// TIA Portal V21 export
FUNCTION_BLOCK "DoFb"   // FB109, LAD
{ S7_Optimized_Access := 'FALSE' }
// stored: AutoNumber false, SetENOAutomatically false
   VAR_INPUT
      sec : Bool;
      AlarmAck : Bool;
      AlwaysTrue : Bool;
      AlwaysFalse : Bool;
      Interlock : Bool;
   END_VAR
   VAR
      Do01 { S7_SetPoint := 'True'} : "DigitalOutput";   // Mm01Cmd
      Do02 { S7_SetPoint := 'True'} : "DigitalOutput";   // Cp01Cmd
      Do03 { S7_SetPoint := 'True'} : "DigitalOutput";   // Htr
      Do04 { S7_SetPoint := 'True'} : "DigitalOutput";   // Lf01
      Do05 { S7_SetPoint := 'True'} : "DigitalOutput";   // DoSpare1
      Do06 { S7_SetPoint := 'True'} : "DigitalOutput";   // DoSpare2
      Do07 { S7_SetPoint := 'True'} : "DigitalOutput";   // DoSpare3
      Do08 { S7_SetPoint := 'True'} : "DigitalOutput";   // DoSpare4
      Do09 { S7_SetPoint := 'True'} : "DigitalOutput";   // DoSpare5
      Do10 { S7_SetPoint := 'True'} : "DigitalOutput";   // DoSpare6
   END_VAR
BEGIN

REGION Network 1: Mm01Cmd
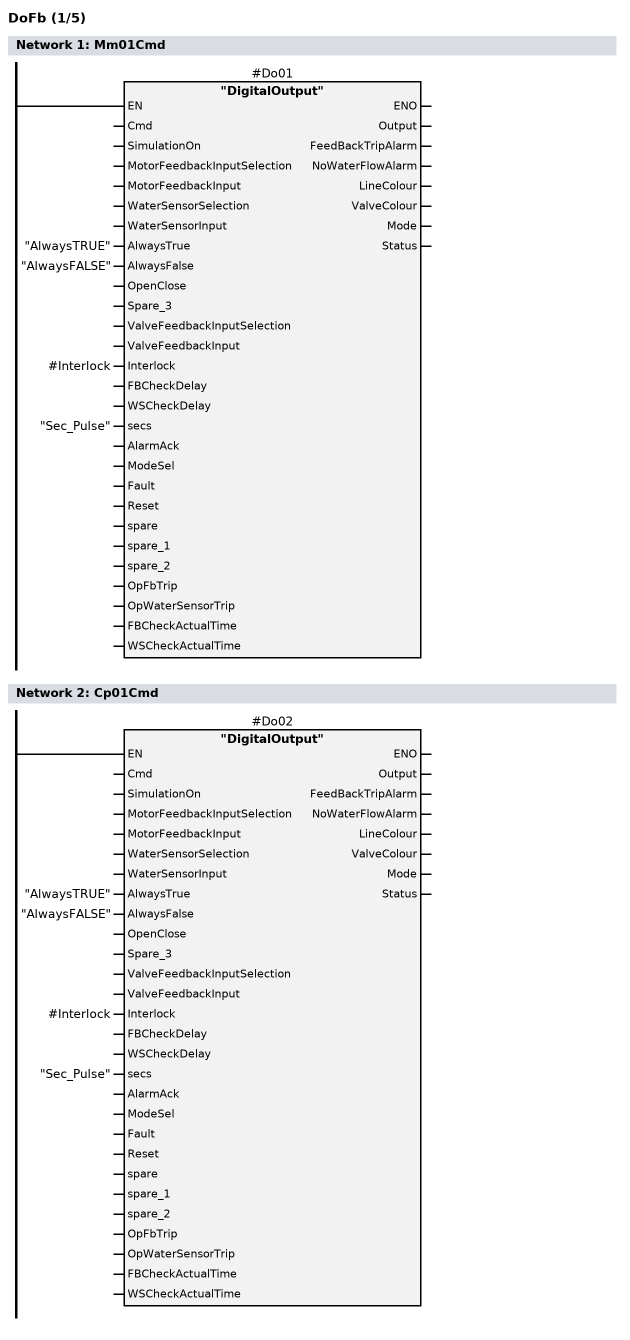
   RUNG wire#powerrail
      #Do01(Cmd :=, SimulationOn :=, MotorFeedbackInputSelection :=, MotorFeedbackInput :=, WaterSensorSelection :=, WaterSensorInput :=, AlwaysTrue := "AlwaysTRUE", AlwaysFalse := "AlwaysFALSE", OpenClose :=, Spare_3 :=, ValveFeedbackInputSelection :=, ValveFeedbackInput :=, Interlock := #Interlock, FBCheckDelay :=, WSCheckDelay :=, secs := "Sec_Pulse", AlarmAck :=, ModeSel :=, Fault :=, Reset :=, spare :=, spare_1 :=, spare_2 :=, OpFbTrip :=, OpWaterSensorTrip :=, FBCheckActualTime :=, WSCheckActualTime :=, Output =>, FeedBackTripAlarm =>, NoWaterFlowAlarm =>, LineColour =>, ValveColour =>, Mode =>, Status =>)
   END_RUNG
   // the same network as SCL:
   #Do01(AlwaysTrue := "AlwaysTRUE", AlwaysFalse := "AlwaysFALSE", Interlock := #Interlock, secs := "Sec_Pulse");   // "DigitalOutput"
END_REGION

REGION Network 2: Cp01Cmd
   RUNG wire#powerrail
      #Do02(Cmd :=, SimulationOn :=, MotorFeedbackInputSelection :=, MotorFeedbackInput :=, WaterSensorSelection :=, WaterSensorInput :=, AlwaysTrue := "AlwaysTRUE", AlwaysFalse := "AlwaysFALSE", OpenClose :=, Spare_3 :=, ValveFeedbackInputSelection :=, ValveFeedbackInput :=, Interlock := #Interlock, FBCheckDelay :=, WSCheckDelay :=, secs := "Sec_Pulse", AlarmAck :=, ModeSel :=, Fault :=, Reset :=, spare :=, spare_1 :=, spare_2 :=, OpFbTrip :=, OpWaterSensorTrip :=, FBCheckActualTime :=, WSCheckActualTime :=, Output =>, FeedBackTripAlarm =>, NoWaterFlowAlarm =>, LineColour =>, ValveColour =>, Mode =>, Status =>)
   END_RUNG
   // the same network as SCL:
   #Do02(AlwaysTrue := "AlwaysTRUE", AlwaysFalse := "AlwaysFALSE", Interlock := #Interlock, secs := "Sec_Pulse");   // "DigitalOutput"
END_REGION

REGION Network 3: Htr
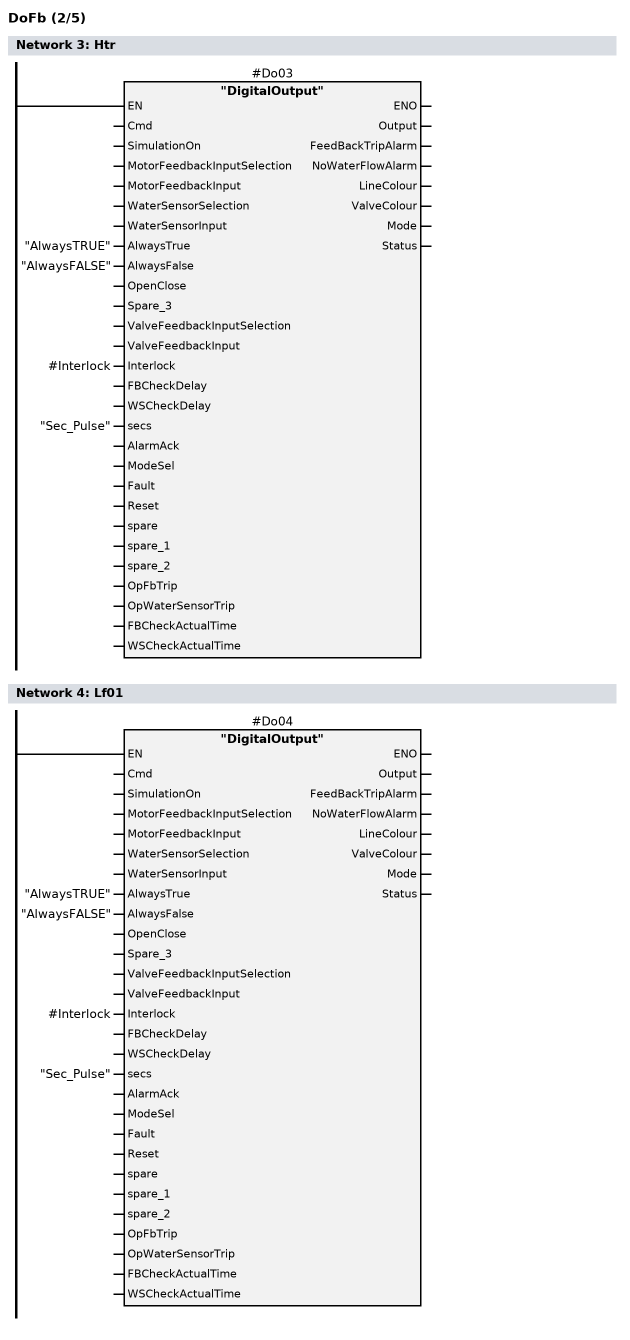
   RUNG wire#powerrail
      #Do03(Cmd :=, SimulationOn :=, MotorFeedbackInputSelection :=, MotorFeedbackInput :=, WaterSensorSelection :=, WaterSensorInput :=, AlwaysTrue := "AlwaysTRUE", AlwaysFalse := "AlwaysFALSE", OpenClose :=, Spare_3 :=, ValveFeedbackInputSelection :=, ValveFeedbackInput :=, Interlock := #Interlock, FBCheckDelay :=, WSCheckDelay :=, secs := "Sec_Pulse", AlarmAck :=, ModeSel :=, Fault :=, Reset :=, spare :=, spare_1 :=, spare_2 :=, OpFbTrip :=, OpWaterSensorTrip :=, FBCheckActualTime :=, WSCheckActualTime :=, Output =>, FeedBackTripAlarm =>, NoWaterFlowAlarm =>, LineColour =>, ValveColour =>, Mode =>, Status =>)
   END_RUNG
   // the same network as SCL:
   #Do03(AlwaysTrue := "AlwaysTRUE", AlwaysFalse := "AlwaysFALSE", Interlock := #Interlock, secs := "Sec_Pulse");   // "DigitalOutput"
END_REGION

REGION Network 4: Lf01
   RUNG wire#powerrail
      #Do04(Cmd :=, SimulationOn :=, MotorFeedbackInputSelection :=, MotorFeedbackInput :=, WaterSensorSelection :=, WaterSensorInput :=, AlwaysTrue := "AlwaysTRUE", AlwaysFalse := "AlwaysFALSE", OpenClose :=, Spare_3 :=, ValveFeedbackInputSelection :=, ValveFeedbackInput :=, Interlock := #Interlock, FBCheckDelay :=, WSCheckDelay :=, secs := "Sec_Pulse", AlarmAck :=, ModeSel :=, Fault :=, Reset :=, spare :=, spare_1 :=, spare_2 :=, OpFbTrip :=, OpWaterSensorTrip :=, FBCheckActualTime :=, WSCheckActualTime :=, Output =>, FeedBackTripAlarm =>, NoWaterFlowAlarm =>, LineColour =>, ValveColour =>, Mode =>, Status =>)
   END_RUNG
   // the same network as SCL:
   #Do04(AlwaysTrue := "AlwaysTRUE", AlwaysFalse := "AlwaysFALSE", Interlock := #Interlock, secs := "Sec_Pulse");   // "DigitalOutput"
END_REGION

REGION Network 5: #Do05 spare1
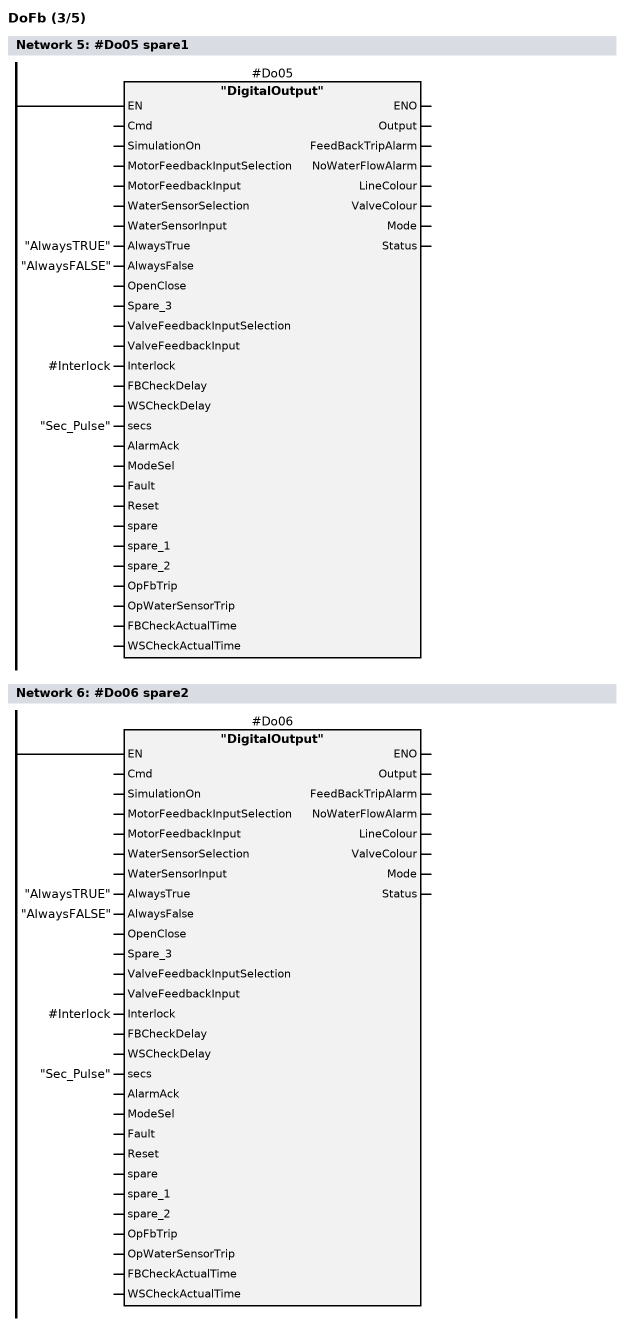
   RUNG wire#powerrail
      #Do05(Cmd :=, SimulationOn :=, MotorFeedbackInputSelection :=, MotorFeedbackInput :=, WaterSensorSelection :=, WaterSensorInput :=, AlwaysTrue := "AlwaysTRUE", AlwaysFalse := "AlwaysFALSE", OpenClose :=, Spare_3 :=, ValveFeedbackInputSelection :=, ValveFeedbackInput :=, Interlock := #Interlock, FBCheckDelay :=, WSCheckDelay :=, secs := "Sec_Pulse", AlarmAck :=, ModeSel :=, Fault :=, Reset :=, spare :=, spare_1 :=, spare_2 :=, OpFbTrip :=, OpWaterSensorTrip :=, FBCheckActualTime :=, WSCheckActualTime :=, Output =>, FeedBackTripAlarm =>, NoWaterFlowAlarm =>, LineColour =>, ValveColour =>, Mode =>, Status =>)
   END_RUNG
   // the same network as SCL:
   #Do05(AlwaysTrue := "AlwaysTRUE", AlwaysFalse := "AlwaysFALSE", Interlock := #Interlock, secs := "Sec_Pulse");   // "DigitalOutput"
END_REGION

REGION Network 6: #Do06 spare2
   RUNG wire#powerrail
      #Do06(Cmd :=, SimulationOn :=, MotorFeedbackInputSelection :=, MotorFeedbackInput :=, WaterSensorSelection :=, WaterSensorInput :=, AlwaysTrue := "AlwaysTRUE", AlwaysFalse := "AlwaysFALSE", OpenClose :=, Spare_3 :=, ValveFeedbackInputSelection :=, ValveFeedbackInput :=, Interlock := #Interlock, FBCheckDelay :=, WSCheckDelay :=, secs := "Sec_Pulse", AlarmAck :=, ModeSel :=, Fault :=, Reset :=, spare :=, spare_1 :=, spare_2 :=, OpFbTrip :=, OpWaterSensorTrip :=, FBCheckActualTime :=, WSCheckActualTime :=, Output =>, FeedBackTripAlarm =>, NoWaterFlowAlarm =>, LineColour =>, ValveColour =>, Mode =>, Status =>)
   END_RUNG
   // the same network as SCL:
   #Do06(AlwaysTrue := "AlwaysTRUE", AlwaysFalse := "AlwaysFALSE", Interlock := #Interlock, secs := "Sec_Pulse");   // "DigitalOutput"
END_REGION

REGION Network 7: #Do07spare3
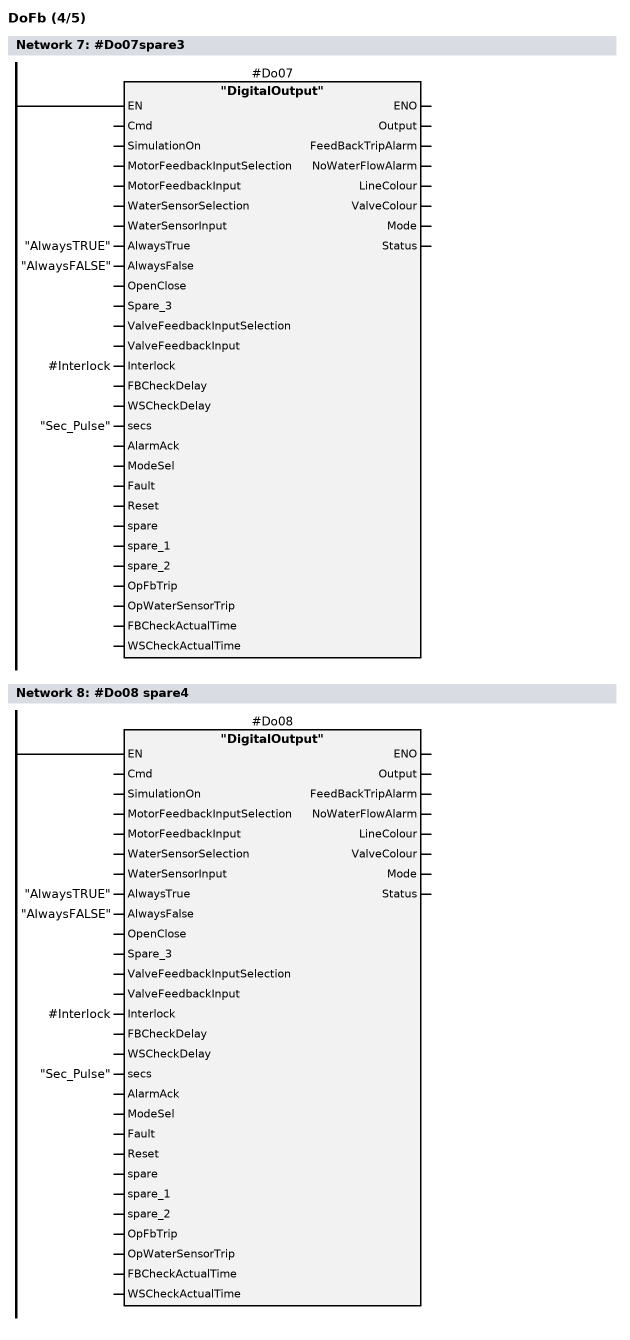
   RUNG wire#powerrail
      #Do07(Cmd :=, SimulationOn :=, MotorFeedbackInputSelection :=, MotorFeedbackInput :=, WaterSensorSelection :=, WaterSensorInput :=, AlwaysTrue := "AlwaysTRUE", AlwaysFalse := "AlwaysFALSE", OpenClose :=, Spare_3 :=, ValveFeedbackInputSelection :=, ValveFeedbackInput :=, Interlock := #Interlock, FBCheckDelay :=, WSCheckDelay :=, secs := "Sec_Pulse", AlarmAck :=, ModeSel :=, Fault :=, Reset :=, spare :=, spare_1 :=, spare_2 :=, OpFbTrip :=, OpWaterSensorTrip :=, FBCheckActualTime :=, WSCheckActualTime :=, Output =>, FeedBackTripAlarm =>, NoWaterFlowAlarm =>, LineColour =>, ValveColour =>, Mode =>, Status =>)
   END_RUNG
   // the same network as SCL:
   #Do07(AlwaysTrue := "AlwaysTRUE", AlwaysFalse := "AlwaysFALSE", Interlock := #Interlock, secs := "Sec_Pulse");   // "DigitalOutput"
END_REGION

REGION Network 8: #Do08 spare4
   RUNG wire#powerrail
      #Do08(Cmd :=, SimulationOn :=, MotorFeedbackInputSelection :=, MotorFeedbackInput :=, WaterSensorSelection :=, WaterSensorInput :=, AlwaysTrue := "AlwaysTRUE", AlwaysFalse := "AlwaysFALSE", OpenClose :=, Spare_3 :=, ValveFeedbackInputSelection :=, ValveFeedbackInput :=, Interlock := #Interlock, FBCheckDelay :=, WSCheckDelay :=, secs := "Sec_Pulse", AlarmAck :=, ModeSel :=, Fault :=, Reset :=, spare :=, spare_1 :=, spare_2 :=, OpFbTrip :=, OpWaterSensorTrip :=, FBCheckActualTime :=, WSCheckActualTime :=, Output =>, FeedBackTripAlarm =>, NoWaterFlowAlarm =>, LineColour =>, ValveColour =>, Mode =>, Status =>)
   END_RUNG
   // the same network as SCL:
   #Do08(AlwaysTrue := "AlwaysTRUE", AlwaysFalse := "AlwaysFALSE", Interlock := #Interlock, secs := "Sec_Pulse");   // "DigitalOutput"
END_REGION

REGION Network 9: ##Do09 spare5
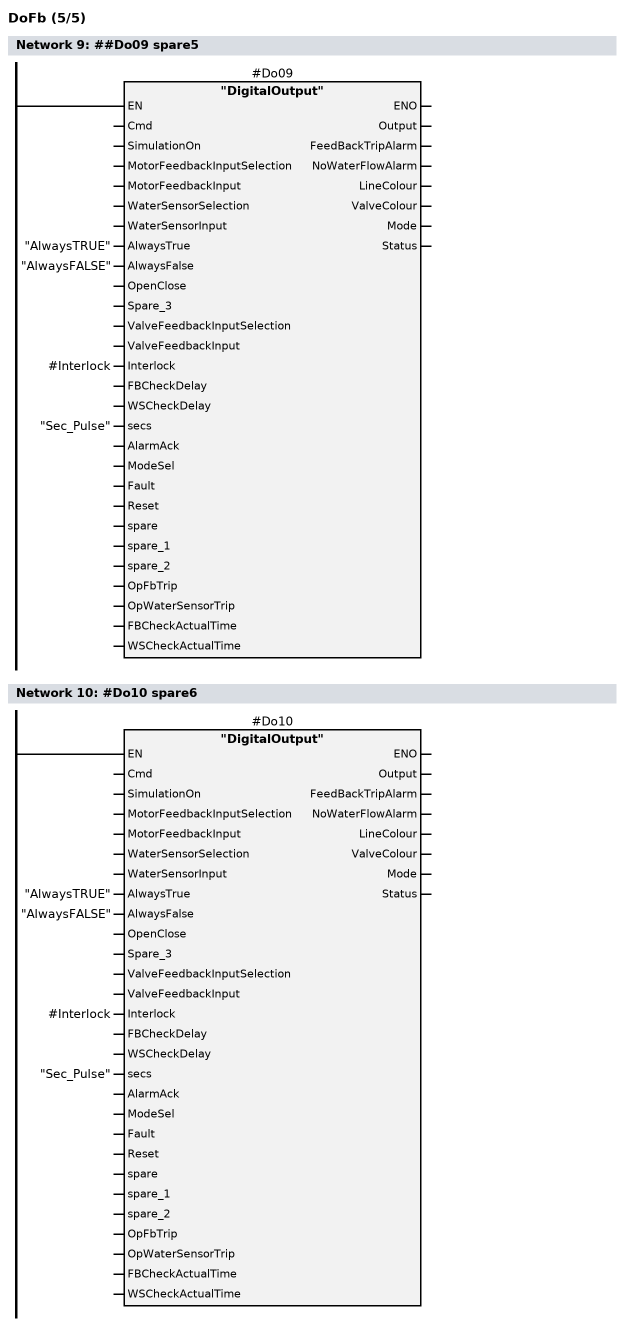
   RUNG wire#powerrail
      #Do09(Cmd :=, SimulationOn :=, MotorFeedbackInputSelection :=, MotorFeedbackInput :=, WaterSensorSelection :=, WaterSensorInput :=, AlwaysTrue := "AlwaysTRUE", AlwaysFalse := "AlwaysFALSE", OpenClose :=, Spare_3 :=, ValveFeedbackInputSelection :=, ValveFeedbackInput :=, Interlock := #Interlock, FBCheckDelay :=, WSCheckDelay :=, secs := "Sec_Pulse", AlarmAck :=, ModeSel :=, Fault :=, Reset :=, spare :=, spare_1 :=, spare_2 :=, OpFbTrip :=, OpWaterSensorTrip :=, FBCheckActualTime :=, WSCheckActualTime :=, Output =>, FeedBackTripAlarm =>, NoWaterFlowAlarm =>, LineColour =>, ValveColour =>, Mode =>, Status =>)
   END_RUNG
   // the same network as SCL:
   #Do09(AlwaysTrue := "AlwaysTRUE", AlwaysFalse := "AlwaysFALSE", Interlock := #Interlock, secs := "Sec_Pulse");   // "DigitalOutput"
END_REGION

REGION Network 10: #Do10 spare6
   RUNG wire#powerrail
      #Do10(Cmd :=, SimulationOn :=, MotorFeedbackInputSelection :=, MotorFeedbackInput :=, WaterSensorSelection :=, WaterSensorInput :=, AlwaysTrue := "AlwaysTRUE", AlwaysFalse := "AlwaysFALSE", OpenClose :=, Spare_3 :=, ValveFeedbackInputSelection :=, ValveFeedbackInput :=, Interlock := #Interlock, FBCheckDelay :=, WSCheckDelay :=, secs := "Sec_Pulse", AlarmAck :=, ModeSel :=, Fault :=, Reset :=, spare :=, spare_1 :=, spare_2 :=, OpFbTrip :=, OpWaterSensorTrip :=, FBCheckActualTime :=, WSCheckActualTime :=, Output =>, FeedBackTripAlarm =>, NoWaterFlowAlarm =>, LineColour =>, ValveColour =>, Mode =>, Status =>)
   END_RUNG
   // the same network as SCL:
   #Do10(AlwaysTrue := "AlwaysTRUE", AlwaysFalse := "AlwaysFALSE", Interlock := #Interlock, secs := "Sec_Pulse");   // "DigitalOutput"
END_REGION
END_FUNCTION_BLOCK
